{attribute 'linkalways'} 
{attribute 'no_explicit_call' := 'This FB is a CLASS and must be accessed using methods or properties'}
{attribute 'enable_dynamic_creation'}
FUNCTION_BLOCK Node_F_VN_ContourElongation EXTENDS VisionNode
VAR
    ipContour : _ITcVnContainer;
    fElongation : _LREAL(0.0);
    hrPrev : _HRESULT(S_OK);
	hresult : _HRESULT(S_OK);
END_VAR

METHOD PUBLIC  Clone : I_Node
VAR
	pNode : POINTER TO Node_F_VN_ContourElongation;
END_VAR
pNode := __NEW(Node_F_VN_ContourElongation);
Clone := pNode^;
END_METHOD

METHOD FB_init : BOOL
VAR_INPUT
	bInitRetains : BOOL; // if TRUE, the retain variables are initialized (warm start / cold start)
	bInCopyCode : BOOL;  // if TRUE, the instance afterwards gets moved into the copy code (online change)
END_VAR
AddInput('ipContour', ipContour);
AddInput('hrPrev', hrPrev);
AddOutput('fElongation', fElongation);
AddOutput('hresult',hresult);
END_METHOD

METHOD PROTECTED OnExecute
hresult.Value := F_VN_ContourElongation(
	ipContour := ipContour.Value,
    fElongation := fElongation.Value,
	hrPrev:= hrPrev.Value);
END_METHOD

METHOD PUBLIC PreExecutionCheck
VAR_INPUT
	Check : I_PreExecutionChecks;
END_VAR
Check.IsTrue(ipContour.IsValid, 'ipContour must be a valid container');
Check.IsTrue((ipContour.IsType(TC_GLOBAL_CONST_LIST.ContainerType_Vector_TcVnPoint2_DINT) OR
              ipContour.IsType(TC_GLOBAL_CONST_LIST.ContainerType_Vector_TcVnPoint2_REAL)),
              'ipContour contains incorrect type');
END_METHOD

END_FUNCTION_BLOCK

(* stored: Version 1.1.0.1, ProductVersion 3.1.4026.13
   POU Node_F_VN_ContourElongation: Id {3dd36538-759d-0da9-2ea2-965c0721f26e}, SpecialFunc None
   Folder Constructor: Id {87b99f2f-6f61-07ff-044a-47746c2741f6}
   Method Clone: Id {34b48934-e4d0-0588-1525-718d2642e4aa}
   Method FB_init: Id {a8129011-ed50-0f93-2c55-26ca06e78478}
   Method OnExecute: Id {4ff31846-ccf9-0568-2b8c-5f2acfe29b57}
   Method PreExecutionCheck: Id {c7d45770-c5f6-0d49-1feb-48367a9676e7} *)
